// TIA Portal project "Groups" (V15.1)

(* hardware
DEVICE "ET 200SP station_1"  ET 200SP-Station
   slot 0: "Rack_0"  Rack  6ES5 710-8MAx1
   slot 1: "-plc"  CPU 1512SP-1 PN  6ES7 512-1DK01-0AB0  V2.5
   slot 2: "Server module_1"  Server module  6ES7 193-6PA00-0AA0  V1.1
      slot 1: "Server module_1"  Server module
   slot 127: "BA 2xRJ45"  BA 2xRJ45  6ES7 193-6AR00-0AA0  V0.0
      slot 32769: "Port_1"  6ES7 193-6AR00-0AA0
      slot 32770: "Port_2"  6ES7 193-6AR00-0AA0
DEVICE "ET 200eco station_1"  ET 200eco station
   slot 0: "Rack_0"  Rail
   slot 0: "-IO device_1"  ET 200eco PN 8DIO  6ES7 147-6BG00-0AB0  V7.0
      slot 1: "8 DIO DC24V/1.3A 8xM12"  6ES7 147-6BG00-0AB0
DEVICE "S71500/ET200MP station_1"  S7-1500 station
   slot 0: "Rail_0"  Rack  6ES7 590-1***0-0AA0
   slot 1: "PLC_1"  CPU 1515-2 PN  6ES7 515-2AM01-0AB0  V2.5
      slot 3: "CPU display_1"  6ES7591-1BA00-0AA0
*)

// ===== PLC "-plc"  CPU 1512SP-1 PN =====

ORGANIZATION_BLOCK "Main"   // OB1, LAD, ProgramCycle
TITLE = "Main Program Sweep (Cycle)"
{ S7_Optimized_Access := 'TRUE' }
VERSION : 0.1
   VAR_INPUT
      Initial_Call : Bool;   // Initial call of this OB
      Remanence : Bool;   // =True, if remanent data are available
   END_VAR
BEGIN
END_ORGANIZATION_BLOCK

// ===== PLC "PLC_1"  CPU 1515-2 PN =====

ORGANIZATION_BLOCK "Main"   // OB1, LAD, ProgramCycle
TITLE = "Main Program Sweep (Cycle)"
{ S7_Optimized_Access := 'TRUE' }
VERSION : 0.1
   VAR_INPUT
      Initial_Call : Bool;   // Initial call of this OB
      Remanence : Bool;   // =True, if remanent data are available
   END_VAR
BEGIN
END_ORGANIZATION_BLOCK